// TIA Portal V18 export
TYPE "FixtureCheck_UDT"
   STRUCT
      FixtureIDSetValue : Int;   // 配方设定的工装ID
      FixtureIDCheckValue : Int;   // 实际检测工装ID
      FixtureCheckResult : Bool;   // 工装检测对比结果，0,NOK; 1,OK
      FixtureCheckUnEnable : Bool;   // 工装检测使能,不需要检测时，给1
   END_STRUCT;
END_TYPE
